TYPE
    PLCopenCallGroupType :
    STRUCT
        _startStep : ENUM; //The step when doStep was called
        _currentStep : ENUM;
        _lastRequestNumber : DINT;
        _onEntry : BOOL;
        _onExit : BOOL;
        _isDone : BOOL;
        _isAbort : BOOL;
        _isError : BOOL;
        _statusChecked : BOOL;
        _numberActiveCommands : INT;
        _commands : ARRAY[0..GVL.MAX_RELATED_GROUPS] OF PLCopenCall;
        _syncAbort : BOOL;
        _syncError : BOOL;
        _syncDone : BOOL;
    END_STRUCT
END_TYPE

(* stored: Version 1.1.0.1
   DUT PLCopenCallGroupType: Id {d3dcb7f9-fdae-4639-b5ca-cb80fdcb3095} *)
